FUNCTION "Int[].CountOfElements" : UDInt
{ S7_Optimized_Access := 'TRUE' }
VERSION : 0.1
   VAR_INPUT
      data : Variant;
   END_VAR


BEGIN
	#"Int[].CountOfElements" := CountOfElements(#data);
	RETURN;
END_FUNCTION

